PROGRAM originRepo2
VAR
END_VAR

END_PROGRAM

(* stored: Version 1.1.0.1, ProductVersion 3.1.4024.12
   POU originRepo2: Id {aaa911db-0e3a-01b3-148d-07ef2642fbc3}, SpecialFunc None *)
